PROGRAM LogicalCircuits_Ex03
VAR
	S2						: DigitalInput_NO;
	P2 						: digitaloutput;
END_VAR

IF S2.isOn THEN
	P2.Off();
ELSE 
	P2.On();
END_IF

END_PROGRAM

(* stored: Version 1.1.0.1
   POU LogicalCircuits_Ex03: Id {e28522be-f6aa-4232-b8ec-b3242f63fad6}, SpecialFunc None *)
